// Implicitly generated code : DO NOT EDIT
FUNCTION CheckBounds : DINT
VAR_INPUT
	index, lower, upper: DINT;
END_VAR

// Implicitly generated code : Only an Implementation suggestion
{noflow}
IF  index < lower THEN
	G_Diag.uiCheckBound:=G_Diag.uiCheckBound+1;
	CheckBounds := lower;
ELSIF  index > upper THEN
	G_Diag.uiCheckBound:=G_Diag.uiCheckBound+1;
	CheckBounds := upper;
ELSE
	CheckBounds := index;
END_IF
{flow}

END_FUNCTION

(* stored: Version 1.1.0.1, ProductVersion 3.1.4024.4
   POU CheckBounds: Id {761e5b1a-c083-47a6-82eb-7a8f20370fb0}, SpecialFunc CheckBounds *)
